// TIA Portal V20 export
DATA_BLOCK "CalcDoseDB_Outlet"   // DB43
// stored: InstanceOfName CalcDose, InstanceOfType FB
"CalcDose"
   // VAR_INPUT
   //    Enable : Bool;
   //    Dose_Liters : Real;
   //    VolumeFlow : Real;
   //    Scale_Raw : "ScaVal_Raw";
   // END_VAR
   // VAR_OUTPUT
   //    Service_Done : Bool;
   //    Liters { ExternalWritable := 'False'} : Real;
   //    Liters_Raw : Real;
   // END_VAR
   // VAR_IN_OUT
   //    AccuSDB : "AccuS";
   // END_VAR
BEGIN
END_DATA_BLOCK
